FUNCTION_BLOCK CoE_property_dint EXTENDS CoE_property
VAR_INPUT
END_VAR
VAR_OUTPUT
END_VAR
VAR
	_value : DINT;
END_VAR

SUPER^();

PROPERTY dataTypeSize : UINT
GET
dataTypeSize := SIZEOF(_value);
END_GET
END_PROPERTY

METHOD get_value : BOOL
VAR_OUTPUT
	value : DINT ;
	errId : UDINT;
END_VAR
IF init_done THEN
	value := _value;
	get_value := TRUE;
ELSE
	errId := 2;
	get_value := FALSE;
END_IF
END_METHOD

METHOD handle_read_callback : BOOL
VAR_INPUT
	pt_buffer : POINTER TO CoE_buffer_type_cast_union;
	errId : UDINT;
END_VAR

_value := pt_buffer^.value_dint;
_init_done:=TRUE;
_read_errId:=errId;
END_METHOD

METHOD set_value : BOOL
VAR_INPUT
	value : dint ;
END_VAR
_valueToWrite.value_dint := value;
IF THIS^._I_CoE_communication_handler <> 0 THEN 
	THIS^._I_CoE_communication_handler.add_write_request(THIS^);
ELSE
	errId:=1;
END_IF
END_METHOD

END_FUNCTION_BLOCK

(* stored: Version 1.1.0.1, ProductVersion 3.1.4024.6
   POU CoE_property_dint: Id {0c5f23ca-29a0-0898-28c5-d1d05d6ed6fc}, SpecialFunc None
   Property dataTypeSize: Id {294e0b5a-1c15-0654-1102-950a709d69b6}
   Get Get: Id {d66eb3b5-4cc8-018e-0769-b103b1a1803f}
   Method get_value: Id {28c6da6f-eba6-008f-1849-f5ec326c74ee}
   Method handle_read_callback: Id {7ff65813-0b7c-02de-1cd7-3d83b5db9a24}
   Method set_value: Id {9e08aa8b-b300-0280-19bb-1f1b21592c90} *)
